// TIA Portal project "SistemRotativCuve_V19" (V19)

(* hardware
DEVICE "ET 200SP station_1"  ET 200SP-Station
   slot 0: "Rack_0"  Rack  6ES5 710-8MAx1
   slot 1: "PLC_1"  CPU 1510SP-1 PN  6ES7 510-1DK03-0AB0  V3.0
      slot 32768: "PROFINET interface_1"  X1
         slot 32771: "Port_3"  X1 P3
   slot 2: "DI 16x24VDC ST_1"  DI 16x24VDC ST  6ES7 131-6BH01-0BA0  V0.0
      slot 1: "DI 16x24VDC ST_1"  DI 16x24VDC ST
   slot 3: "DQ 16x24VDC/0.5A ST_1"  DQ 16x24VDC/0.5A ST  6ES7 132-6BH01-0BA0  V0.0
      slot 1: "DQ 16x24VDC/0.5A ST_1"  DQ 16x24VDC/0.5A ST
   slot 4: "Server module_1"  Server module  6ES7 193-6PA00-0AA0  V1.1
      slot 1: "Server module_1"  Server module
   slot 127: "BA 2xRJ45"  BA 2xRJ45  6ES7 193-6AR00-0AA0  V0.0
      slot 32769: "Port_1"  X1 P1  6ES7 193-6AR00-0AA0
      slot 32770: "Port_2"  X1 P2  6ES7 193-6AR00-0AA0
DEVICE "HMI_2"  KTP1200 Basic PN
   slot 0: "HMI_2"  KTP1200 Basic PN  6AV2 123-2MB03-0AX0  17.0.0.0
   slot 1: "HMI_RT_2"  KTP1200 Basic PN  6AV2 123-2MB03-0AX0  17.0.0.0
   slot 5: "HMI_2.IE_CP_1"  PROFINET Interface  17.0.0.0
      slot 1: "PROFINET Interface_1"  PROFINET Interface
         slot 1: "Port_1"  Port
*)

// ===== PLC "PLC_1"  CPU 1510SP-1 PN =====

VAR_GLOBAL   // PLC tag table "Default tag table"
   "System_Byte" AT %MB1 : Byte;
   "FirstScan" AT %M1.0 : Bool;
   "DiagStatusUpdate" AT %M1.1 : Bool;
   "AlwaysTRUE" AT %M1.2 : Bool;
   "AlwaysFALSE" AT %M1.3 : Bool;
END_VAR

VAR_GLOBAL   // PLC tag table "Clock Memory"
   "Clock_Byte" AT %MB0 : Byte;
   "Clock_10Hz" AT %M0.0 : Bool;
   "Clock_5Hz" AT %M0.1 : Bool;
   "Clock_2.5Hz" AT %M0.2 : Bool;
   "Clock_2Hz" AT %M0.3 : Bool;
   "Clock_1.25Hz" AT %M0.4 : Bool;
   "Clock_1Hz" AT %M0.5 : Bool;
   "Clock_0.625Hz" AT %M0.6 : Bool;
   "Clock_0.5Hz" AT %M0.7 : Bool;
END_VAR

VAR_GLOBAL   // PLC tag table "Motor_Tags"
   "Motor_Start" AT %M4.1 : Bool;
   "Motor_Stop" AT %M4.2 : Bool;
   "Motor_Ready_to_Start" AT %M4.3 : Bool;
END_VAR

VAR_GLOBAL   // PLC tag table "Sensors_Tags"
   "Barrier_Detection_Sensor1" AT %M3.0 : Bool;
   "Filling_Box_Sensor1" AT %M3.1 : Bool;
   "Emptying_Box_Sensor2" AT %M3.2 : Bool;
   "Barrier_Detection_Time_ON" AT %QD3 : DInt;
END_VAR

VAR_GLOBAL   // PLC tag table "Conveyor_Tags"
   "Conveyor_Start" AT %M5.1 : Bool;
   "Conveyor_Stop" AT %M5.2 : Bool;
   "Conveyor_Ready_to_Start" AT %M5.3 : Bool;
END_VAR

VAR_GLOBAL   // PLC tag table "Buttons"
   "Reset_Rotation_Counter" AT %M2.3 : Bool;
   "Switch_Manual_Mode_Position" AT %M2.4 : Bool;
   "One_Rotation_Move_Button" AT %M2.5 : Bool;
   "Switch_Automatic_Mode_Position" AT %M2.6 : Bool;
   "Switch_Stop_Mode_Position" AT %M2.7 : Bool;
END_VAR

VAR_GLOBAL   // PLC tag table "States"
   "Filled_All_Boxes" AT %M1.6 : Bool;
   "General_Stop_All_Filled" AT %M2.0 : Bool;
   "Automatic_Mode_ON" AT %M1.7 : Bool;
   "Manual_Mode_ON" AT %M2.1 : Bool;
   "General_Stop_Mode_ON" AT %M2.2 : Bool;
END_VAR

// folder: Conveyor/Data_Blocks

DATA_BLOCK "Conveyor_Drive_DB"   // DB4
{ S7_Optimized_Access := 'TRUE' }
VERSION : 0.1
// stored: InstanceOfName Conveyor_Drive_FB
"Conveyor_Drive_FB"
BEGIN
END_DATA_BLOCK

// folder: Motor/Data_Blocks

DATA_BLOCK "Counter_Box_Rotation_DB"   // DB2
{ S7_Optimized_Access := 'TRUE' }
AUTHOR : Simatic
FAMILY : IEC
NAME : CNTR
VERSION : 1.0
// stored: InstanceOfName IEC_COUNTER
"IEC_COUNTER"
BEGIN
END_DATA_BLOCK

DATA_BLOCK "Motor_Drive_DB"   // DB3
{ S7_Optimized_Access := 'TRUE' }
VERSION : 0.1
// stored: InstanceOfName Motor_Drive_FB
"Motor_Drive_FB"
BEGIN
END_DATA_BLOCK

// folder: Sensors/Data_Blocks

DATA_BLOCK "Validate_by_Sensors_DB"   // DB1
{ S7_Optimized_Access := 'TRUE' }
VERSION : 0.1
// stored: InstanceOfName Validate_by_Sensors_FB
"Validate_by_Sensors_FB"
BEGIN
END_DATA_BLOCK

DATA_BLOCK "IEC_Timer_0_DB"   // DB8
{ S7_Optimized_Access := 'TRUE' }
AUTHOR : Simatic
FAMILY : IEC
NAME : IEC_TMR
VERSION : 1.0
// stored: InstanceOfName IEC_TIMER
"IEC_TIMER"
BEGIN
END_DATA_BLOCK

// folder: Work Mode/Data_Blocks

DATA_BLOCK "Atomatic_Mode_DB"   // DB5
{ S7_Optimized_Access := 'TRUE' }
VERSION : 0.1
// stored: InstanceOfName Atomatic_Mode_FB
"Atomatic_Mode_FB"
BEGIN
END_DATA_BLOCK

DATA_BLOCK "Manual_Mode_DB"   // DB6
{ S7_Optimized_Access := 'TRUE' }
VERSION : 0.1
// stored: InstanceOfName Manual_Mode_FB
"Manual_Mode_FB"
BEGIN
END_DATA_BLOCK

DATA_BLOCK "General_Stop_Mode_DB"   // DB7
{ S7_Optimized_Access := 'TRUE' }
VERSION : 0.1
// stored: InstanceOfName General_Stop_Mode_FB
"General_Stop_Mode_FB"
BEGIN
END_DATA_BLOCK

// folder: (top level)

ORGANIZATION_BLOCK "Main"   // OB1, LAD, ProgramCycle
TITLE = "Main Program Sweep (Cycle)"
{ S7_Optimized_Access := 'TRUE' }
VERSION : 0.1
// Proiect realizat de Octavian Duma
   VAR_INPUT
      Initial_Call : Bool;   // Initial call of this OB
      Remanence : Bool;   // =True, if remanent data are available
   END_VAR
BEGIN

REGION Network 1: Automatic Mode enabled
   // Aici e scrisa logica de intrare in mod automat prin butonul cu 3 pozitii, setat pe pozitia de mod automat
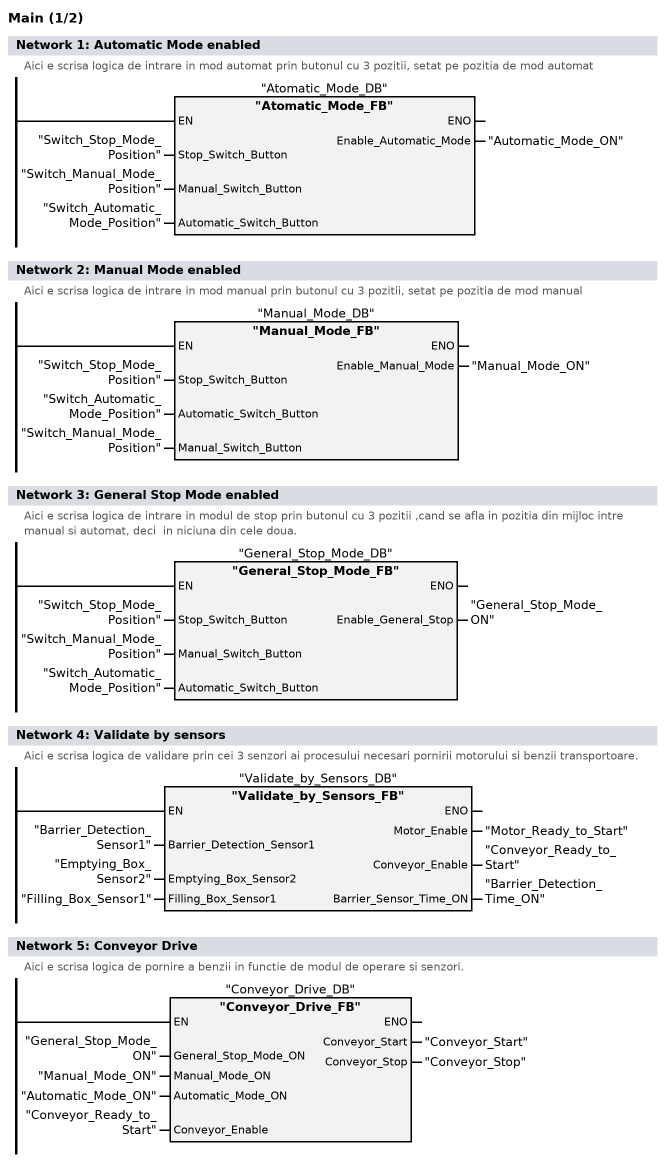
   RUNG wire#powerrail
      "Atomatic_Mode_DB"(Stop_Switch_Button := "Switch_Stop_Mode_Position", Manual_Switch_Button := "Switch_Manual_Mode_Position", Automatic_Switch_Button := "Switch_Automatic_Mode_Position", Enable_Automatic_Mode => "Automatic_Mode_ON")
   END_RUNG
   // the same network as SCL:
   "Atomatic_Mode_DB"(Stop_Switch_Button := "Switch_Stop_Mode_Position",   // "Atomatic_Mode_FB"
                      Manual_Switch_Button := "Switch_Manual_Mode_Position",
                      Automatic_Switch_Button := "Switch_Automatic_Mode_Position",
                      Enable_Automatic_Mode => "Automatic_Mode_ON");
END_REGION

REGION Network 2: Manual Mode enabled
   // Aici e scrisa logica de intrare in mod manual prin butonul cu 3 pozitii, setat pe pozitia de mod manual
   RUNG wire#powerrail
      "Manual_Mode_DB"(Stop_Switch_Button := "Switch_Stop_Mode_Position", Automatic_Switch_Button := "Switch_Automatic_Mode_Position", Manual_Switch_Button := "Switch_Manual_Mode_Position", Enable_Manual_Mode => "Manual_Mode_ON")
   END_RUNG
   // the same network as SCL:
   "Manual_Mode_DB"(Stop_Switch_Button := "Switch_Stop_Mode_Position",   // "Manual_Mode_FB"
                    Automatic_Switch_Button := "Switch_Automatic_Mode_Position",
                    Manual_Switch_Button := "Switch_Manual_Mode_Position",
                    Enable_Manual_Mode => "Manual_Mode_ON");
END_REGION

REGION Network 3: General Stop Mode enabled
   // Aici e scrisa logica de intrare in modul de stop prin butonul cu 3 pozitii ,cand se afla in pozitia din mijloc intre manual si automat, deci  in niciuna din cele doua.
   RUNG wire#powerrail
      "General_Stop_Mode_DB"(Stop_Switch_Button := "Switch_Stop_Mode_Position", Manual_Switch_Button := "Switch_Manual_Mode_Position", Automatic_Switch_Button := "Switch_Automatic_Mode_Position", Enable_General_Stop => "General_Stop_Mode_ON")
   END_RUNG
   // the same network as SCL:
   "General_Stop_Mode_DB"(Stop_Switch_Button := "Switch_Stop_Mode_Position",   // "General_Stop_Mode_FB"
                          Manual_Switch_Button := "Switch_Manual_Mode_Position",
                          Automatic_Switch_Button := "Switch_Automatic_Mode_Position",
                          Enable_General_Stop => "General_Stop_Mode_ON");
END_REGION

REGION Network 4: Validate by sensors
   // Aici e scrisa logica de validare prin cei 3 senzori ai procesului necesari pornirii motorului si benzii transportoare.
   RUNG wire#powerrail
      "Validate_by_Sensors_DB"(Barrier_Detection_Sensor1 := "Barrier_Detection_Sensor1", Emptying_Box_Sensor2 := "Emptying_Box_Sensor2", Filling_Box_Sensor1 := "Filling_Box_Sensor1", Motor_Enable => "Motor_Ready_to_Start", Conveyor_Enable => "Conveyor_Ready_to_Start", Barrier_Sensor_Time_ON => "Barrier_Detection_Time_ON")
   END_RUNG
   // the same network as SCL:
   "Validate_by_Sensors_DB"(Barrier_Detection_Sensor1 := "Barrier_Detection_Sensor1",   // "Validate_by_Sensors_FB"
                           Emptying_Box_Sensor2 := "Emptying_Box_Sensor2",
                           Filling_Box_Sensor1 := "Filling_Box_Sensor1",
                           Motor_Enable => "Motor_Ready_to_Start",
                           Conveyor_Enable => "Conveyor_Ready_to_Start",
                           Barrier_Sensor_Time_ON => "Barrier_Detection_Time_ON");
END_REGION

REGION Network 5: Conveyor Drive
   // Aici e scrisa logica de pornire a benzii in functie de modul de operare si senzori.
   RUNG wire#powerrail
      "Conveyor_Drive_DB"(General_Stop_Mode_ON := "General_Stop_Mode_ON", Manual_Mode_ON := "Manual_Mode_ON", Automatic_Mode_ON := "Automatic_Mode_ON", Conveyor_Enable := "Conveyor_Ready_to_Start", Conveyor_Start => "Conveyor_Start", Conveyor_Stop => "Conveyor_Stop")
   END_RUNG
   // the same network as SCL:
   "Conveyor_Drive_DB"(General_Stop_Mode_ON := "General_Stop_Mode_ON",   // "Conveyor_Drive_FB"
                       Manual_Mode_ON := "Manual_Mode_ON",
                       Automatic_Mode_ON := "Automatic_Mode_ON",
                       Conveyor_Enable := "Conveyor_Ready_to_Start",
                       Conveyor_Start => "Conveyor_Start",
                       Conveyor_Stop => "Conveyor_Stop");
END_REGION

REGION Network 6: Motor Drive
   // Aici e scrisa logica de pornire a motorului in functie de modul de operare, senzori, precum si cazul in care sistemul este plin complet si se goleste la buton in modul manual.
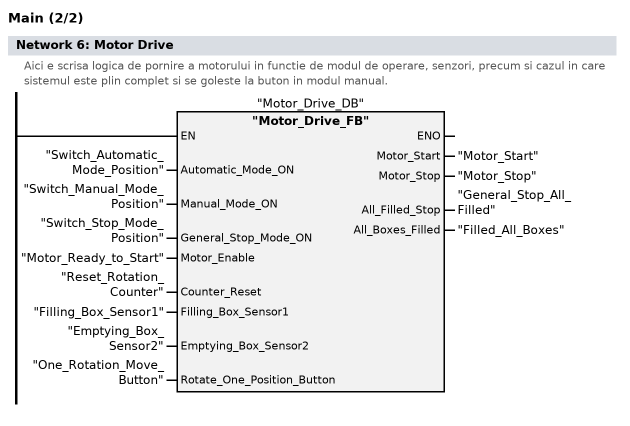
   RUNG wire#powerrail
      "Motor_Drive_DB"(Automatic_Mode_ON := "Switch_Automatic_Mode_Position", Manual_Mode_ON := "Switch_Manual_Mode_Position", General_Stop_Mode_ON := "Switch_Stop_Mode_Position", Motor_Enable := "Motor_Ready_to_Start", Counter_Reset := "Reset_Rotation_Counter", Filling_Box_Sensor1 := "Filling_Box_Sensor1", Emptying_Box_Sensor2 := "Emptying_Box_Sensor2", Rotate_One_Position_Button := "One_Rotation_Move_Button", Motor_Start => "Motor_Start", Motor_Stop => "Motor_Stop", All_Filled_Stop => "General_Stop_All_Filled", All_Boxes_Filled => "Filled_All_Boxes")
   END_RUNG
   // the same network as SCL:
   "Motor_Drive_DB"(Automatic_Mode_ON := "Switch_Automatic_Mode_Position",   // "Motor_Drive_FB"
                    Manual_Mode_ON := "Switch_Manual_Mode_Position",
                    General_Stop_Mode_ON := "Switch_Stop_Mode_Position",
                    Motor_Enable := "Motor_Ready_to_Start",
                    Counter_Reset := "Reset_Rotation_Counter",
                    Filling_Box_Sensor1 := "Filling_Box_Sensor1",
                    Emptying_Box_Sensor2 := "Emptying_Box_Sensor2",
                    Rotate_One_Position_Button := "One_Rotation_Move_Button",
                    Motor_Start => "Motor_Start",
                    Motor_Stop => "Motor_Stop",
                    All_Filled_Stop => "General_Stop_All_Filled",
                    All_Boxes_Filled => "Filled_All_Boxes");
END_REGION
END_ORGANIZATION_BLOCK

// folder: Conveyor/FunctionsDB

FUNCTION_BLOCK "Conveyor_Drive_FB"   // FB2, LAD
{ S7_Optimized_Access := 'TRUE' }
VERSION : 0.1
   VAR_INPUT
      General_Stop_Mode_ON : Bool;
      Manual_Mode_ON : Bool;
      Automatic_Mode_ON : Bool;
      Conveyor_Enable : Bool;
   END_VAR
   VAR_OUTPUT
      Conveyor_Start : Bool;
      Conveyor_Stop : Bool;
   END_VAR
BEGIN

REGION Network 1: Automatic Mode Conveyor is started
   // Banda este pornita in modul automat cand primeste semnalul de enable de la senzori.
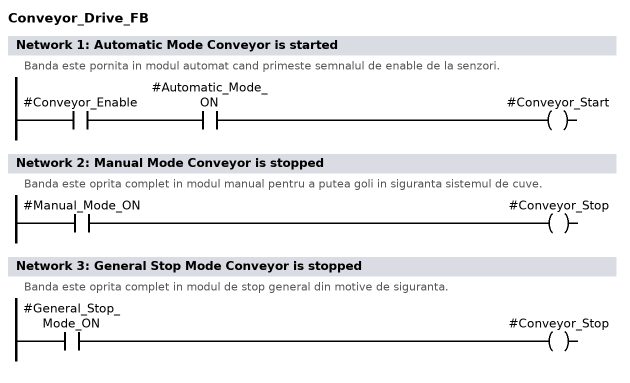
   RUNG wire#powerrail
      Contact( #Conveyor_Enable )
      Contact( #Automatic_Mode_ON )
      Coil( #Conveyor_Start )
   END_RUNG
   // the same network as SCL:
   #Conveyor_Start := #Conveyor_Enable AND #Automatic_Mode_ON;
END_REGION

REGION Network 2: Manual Mode Conveyor is stopped
   // Banda este oprita complet in modul manual pentru a putea goli in siguranta sistemul de cuve.
   RUNG wire#powerrail
      Contact( #Manual_Mode_ON )
      Coil( #Conveyor_Stop )
   END_RUNG
   // the same network as SCL:
   #Conveyor_Stop := #Manual_Mode_ON;
END_REGION

REGION Network 3: General Stop Mode Conveyor is stopped
   // Banda este oprita complet in modul de stop general din motive de siguranta.
   RUNG wire#powerrail
      Contact( #General_Stop_Mode_ON )
      Coil( #Conveyor_Stop )
   END_RUNG
   // the same network as SCL:
   #Conveyor_Stop := #General_Stop_Mode_ON;
END_REGION
END_FUNCTION_BLOCK

// folder: Motor/FunctionsDB

FUNCTION_BLOCK "Motor_Drive_FB"   // FB3, LAD
{ S7_Optimized_Access := 'TRUE' }
VERSION : 0.1
   VAR_INPUT
      Automatic_Mode_ON : Bool;
      Manual_Mode_ON : Bool;
      General_Stop_Mode_ON : Bool;
      Motor_Enable : Bool;
      Counter_Reset : Bool;
      Filling_Box_Sensor1 : Bool;
      Emptying_Box_Sensor2 : Bool;
      Rotate_One_Position_Button : Bool;
   END_VAR
   VAR_OUTPUT
      Motor_Start : Bool;
      Motor_Stop : Bool;
      All_Filled_Stop : Bool;
      All_Boxes_Filled : Bool;
   END_VAR
   VAR
      Rotation_Command : Bool;
   END_VAR
BEGIN

REGION Network 1: Manual Mode Rotation Command
   // Comanda de rotire manuala cu cate o pozitie a cuvei este conditionata de modul manual si de apasarea butonului fizic de pe panoul de comanda.
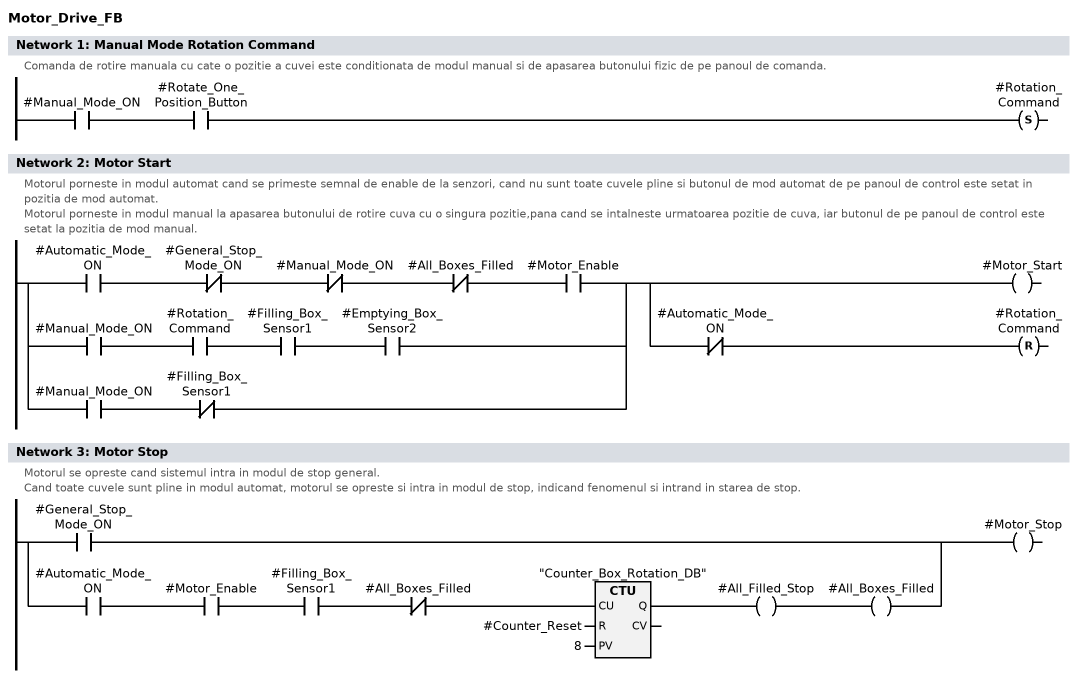
   RUNG wire#powerrail
      Contact( #Manual_Mode_ON )
      Contact( #Rotate_One_Position_Button )
      S_Coil( #Rotation_Command )
   END_RUNG
   // the same network as SCL:
   IF #Manual_Mode_ON AND #Rotate_One_Position_Button THEN #Rotation_Command := TRUE; END_IF;
END_REGION

REGION Network 2: Motor Start
   // Motorul porneste in modul automat cand se primeste semnal de enable de la senzori, cand nu sunt toate cuvele pline si butonul de mod automat de pe panoul de control este setat in pozitia de mod automat. 
   //       Motorul porneste in modul manual la apasarea butonului de rotire cuva cu o singura pozitie,pana cand se intalneste urmatoarea pozitie de cuva, iar butonul de pe panoul de control este setat la pozitia de mod manual.
   RUNG wire#powerrail
      Contact( #Automatic_Mode_ON )
      I_Contact( #General_Stop_Mode_ON )
      I_Contact( #Manual_Mode_ON )
      I_Contact( #All_Boxes_Filled )
      Contact( #Motor_Enable )
      wire#w1
      Coil( #Motor_Start )
   END_RUNG
   RUNG wire#powerrail
      Contact( #Manual_Mode_ON )
      Contact( #Rotation_Command )
      Contact( #Filling_Box_Sensor1 )
      Contact( #Emptying_Box_Sensor2 )
   END_RUNG wire#w1
   RUNG wire#powerrail
      Contact( #Manual_Mode_ON )
      I_Contact( #Filling_Box_Sensor1 )
   END_RUNG wire#w1
   RUNG wire#w1
      I_Contact( #Automatic_Mode_ON )
      R_Coil( #Rotation_Command )
   END_RUNG
   // the same network as SCL:
   #Motor_Start := (#Automatic_Mode_ON AND NOT #General_Stop_Mode_ON AND NOT #Manual_Mode_ON AND NOT #All_Boxes_Filled AND #Motor_Enable) OR (#Manual_Mode_ON AND #Rotation_Command AND #Filling_Box_Sensor1 AND #Emptying_Box_Sensor2) OR (#Manual_Mode_ON AND NOT #Filling_Box_Sensor1);
   IF #Motor_Start AND NOT #Automatic_Mode_ON THEN #Rotation_Command := FALSE; END_IF;
END_REGION

REGION Network 3: Motor Stop
   // Motorul se opreste cand sistemul intra in modul de stop general.
   // Cand toate cuvele sunt pline in modul automat, motorul se opreste si intra in modul de stop, indicand fenomenul si intrand in starea de stop.
   "Counter_Box_Rotation_DB".CTU(CU := #Automatic_Mode_ON AND #Motor_Enable AND #Filling_Box_Sensor1 AND NOT #All_Boxes_Filled,
                           R := #Counter_Reset,
                           PV := 8);
   #All_Filled_Stop := "Counter_Box_Rotation_DB".Q;
   #All_Boxes_Filled := "Counter_Box_Rotation_DB".Q;
   #Motor_Stop := #General_Stop_Mode_ON OR "Counter_Box_Rotation_DB".Q;
END_REGION
END_FUNCTION_BLOCK

// folder: Sensors/FunctionsDB

FUNCTION_BLOCK "Validate_by_Sensors_FB"   // FB1, LAD
{ S7_Optimized_Access := 'TRUE' }
VERSION : 0.1
   VAR_INPUT
      Barrier_Detection_Sensor1 : Bool;
      Emptying_Box_Sensor2 : Bool;
      Filling_Box_Sensor1 : Bool;
   END_VAR
   VAR_OUTPUT
      Motor_Enable : Bool;
      Conveyor_Enable : Bool;
      Barrier_Sensor_Time_ON : DInt;
   END_VAR
   VAR
      Filled_Box : Bool;
   END_VAR
BEGIN

REGION Network 1: A box is full when barrier sensor is ON for 5 seconds
   // Logica de verificare a semnalului senzorului. Pentru a evita activarea conditiei de cuva plina de catre suruburile care cad in cuva de pe banda, senzorul va trebui sa fie activ cel putin 5 secunde ca sa consideram atingerea nivelului de umplere.
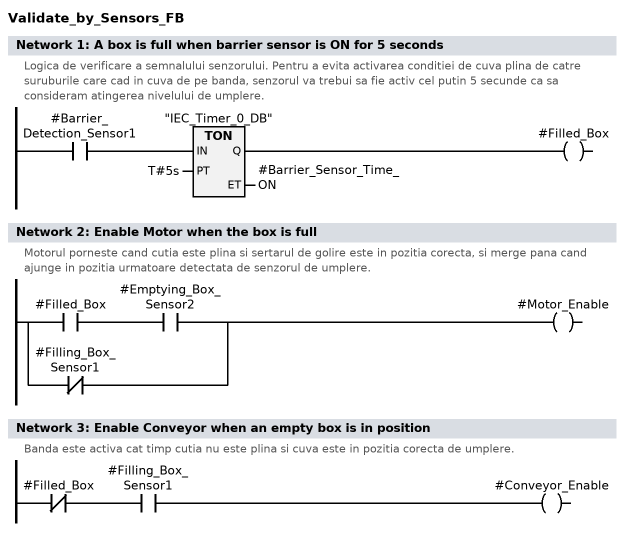
   "IEC_Timer_0_DB".TON(IN := #Barrier_Detection_Sensor1, PT := T#5s, ET => #Barrier_Sensor_Time_ON);
   #Filled_Box := "IEC_Timer_0_DB".Q;
END_REGION

REGION Network 2: Enable Motor when the box is full
   // Motorul porneste cand cutia este plina si sertarul de golire este in pozitia corecta, si merge pana cand ajunge in pozitia urmatoare detectata de senzorul de umplere.
   RUNG wire#powerrail
      Contact( #Filled_Box )
      Contact( #Emptying_Box_Sensor2 )
      wire#w1
      Coil( #Motor_Enable )
   END_RUNG
   RUNG wire#powerrail
      I_Contact( #Filling_Box_Sensor1 )
   END_RUNG wire#w1
   // the same network as SCL:
   #Motor_Enable := (#Filled_Box AND #Emptying_Box_Sensor2) OR NOT #Filling_Box_Sensor1;
END_REGION

REGION Network 3: Enable Conveyor when an empty box is in position
   // Banda este activa cat timp cutia nu este plina si cuva este in pozitia corecta de umplere.
   RUNG wire#powerrail
      I_Contact( #Filled_Box )
      Contact( #Filling_Box_Sensor1 )
      Coil( #Conveyor_Enable )
   END_RUNG
   // the same network as SCL:
   #Conveyor_Enable := NOT #Filled_Box AND #Filling_Box_Sensor1;
END_REGION
END_FUNCTION_BLOCK

// folder: Work Mode/FunctionsDB

FUNCTION_BLOCK "Atomatic_Mode_FB"   // FB4, LAD
{ S7_Optimized_Access := 'TRUE' }
VERSION : 0.1
   VAR_INPUT
      Stop_Switch_Button : Bool;
      Manual_Switch_Button : Bool;
      Automatic_Switch_Button : Bool;
   END_VAR
   VAR_OUTPUT
      Enable_Automatic_Mode : Bool;
   END_VAR
BEGIN

REGION Network 1: Enable Automatic Mode while other mode is disabled
   // Sistemul intra in modul automat pe baza switch-ului cu 3 pozitii, care va fi doar pe pozitia de mod automat , implicand ca celelalte pozitii sa fie dezactivate. Se tine cont si de faptul ca sistemul nu este oprit de umplerea tuturor cuvelor.
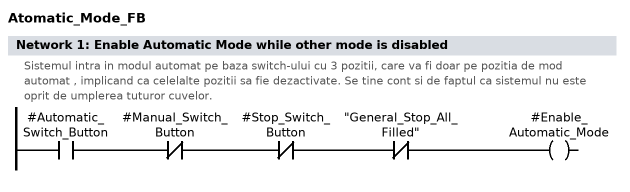
   RUNG wire#powerrail
      Contact( #Automatic_Switch_Button )
      I_Contact( #Manual_Switch_Button )
      I_Contact( #Stop_Switch_Button )
      I_Contact( "General_Stop_All_Filled" )
      Coil( #Enable_Automatic_Mode )
   END_RUNG
   // the same network as SCL:
   #Enable_Automatic_Mode := #Automatic_Switch_Button AND NOT #Manual_Switch_Button AND NOT #Stop_Switch_Button AND NOT "General_Stop_All_Filled";
END_REGION
END_FUNCTION_BLOCK

FUNCTION_BLOCK "Manual_Mode_FB"   // FB5, LAD
{ S7_Optimized_Access := 'TRUE' }
VERSION : 0.1
   VAR_INPUT
      Stop_Switch_Button : Bool;
      Automatic_Switch_Button : Bool;
      Manual_Switch_Button : Bool;
   END_VAR
   VAR_OUTPUT
      Enable_Manual_Mode : Bool;
   END_VAR
BEGIN

REGION Network 1: Enable Manual Mode while other mode is disabled
   // Sistemul intra in modul manual pe baza switch-ului cu 3 pozitii, care va fi doar pe pozitia de mod manual , implicand ca celelalte pozitii sa fie dezactivate. Se tine cont si de faptul ca sistemul nu este oprit de umplerea tuturor cuvelor.
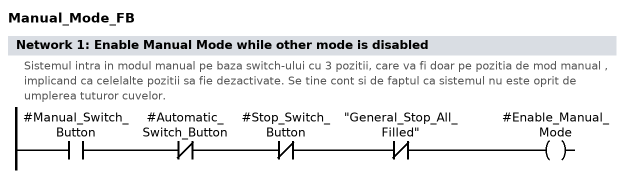
   RUNG wire#powerrail
      Contact( #Manual_Switch_Button )
      I_Contact( #Automatic_Switch_Button )
      I_Contact( #Stop_Switch_Button )
      I_Contact( "General_Stop_All_Filled" )
      Coil( #Enable_Manual_Mode )
   END_RUNG
   // the same network as SCL:
   #Enable_Manual_Mode := #Manual_Switch_Button AND NOT #Automatic_Switch_Button AND NOT #Stop_Switch_Button AND NOT "General_Stop_All_Filled";
END_REGION
END_FUNCTION_BLOCK

FUNCTION_BLOCK "General_Stop_Mode_FB"   // FB6, LAD
{ S7_Optimized_Access := 'TRUE' }
VERSION : 0.1
   VAR_INPUT
      Stop_Switch_Button : Bool;
      Manual_Switch_Button : Bool;
      Automatic_Switch_Button : Bool;
   END_VAR
   VAR_OUTPUT
      Enable_General_Stop : Bool;
   END_VAR
BEGIN

REGION Network 1: Enable General Stop Mode while other mode is disabled
   // Sistemul intra in modul automat pe baza switch-ului cu 3 pozitii, care va fi doar pe pozitia de mod general de stop, fiind pozitia de la mijloc,intre celelate moduri , implicand ca celelalte pozitii sa fie dezactivate.
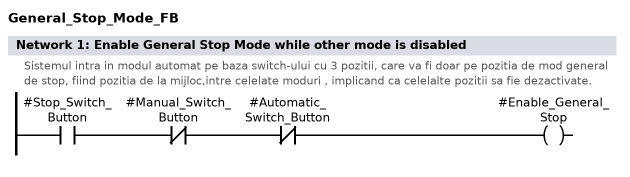
   RUNG wire#powerrail
      Contact( #Stop_Switch_Button )
      I_Contact( #Manual_Switch_Button )
      I_Contact( #Automatic_Switch_Button )
      Coil( #Enable_General_Stop )
   END_RUNG
   // the same network as SCL:
   #Enable_General_Stop := #Stop_Switch_Button AND NOT #Manual_Switch_Button AND NOT #Automatic_Switch_Button;
END_REGION
END_FUNCTION_BLOCK

(* ===== HMI "HMI_RT_2" =====
system functions are stored by id; their names below are inferred from use
connection "HMI_Connection_2": ETHERNET, SMART_S7_1500_OMS

HMI tags "Default tag table"
   "Tag_ScreenNumber" : UInt, internal
   "BarrierDetectionSensor1" : Bool = PLC Barrier_Detection_Sensor1 AT %M3.0, 1 s
   "Conveyor_Ready_to_Start" : Bool = PLC Conveyor_Ready_to_Start AT %M5.3, 1 s
   "Conveyor_Start" : Bool = PLC Conveyor_Start AT %M5.1, 1 s
   "Conveyor_Stop" : Bool = PLC Conveyor_Stop AT %M5.2, 1 s
   "EmptyingBoxSensor2" : Bool = PLC Emptying_Box_Sensor2 AT %M3.2, 1 s
   "FillingBoxSensor1" : Bool = PLC Filling_Box_Sensor1 AT %M3.1, 1 s
   "General_Stop_All_Filled" : Bool = PLC General_Stop_All_Filled AT %M2.0, 1 s
   "Motor_Ready_to_Start" : Bool = PLC Motor_Ready_to_Start AT %M4.3, 1 s
   "Motor_Start" : Bool = PLC Motor_Start AT %M4.1, 1 s
   "Motor_Stop" : Bool = PLC Motor_Stop AT %M4.2, 1 s
   "Reset_Rotation_Counter" : Bool = PLC Reset_Rotation_Counter AT %M2.3, 1 s
   "Rotation_Counter" : Int = PLC Counter_Box_Rotation_DB.CV AT %DB1.DBX0.0, 1 s
   "System_Full" : Bool = PLC Filled_All_Boxes AT %M1.6, 1 s
   "Automatic_Mode_Switch_Position" : Bool = PLC Switch_Automatic_Mode_Position AT %M2.6, 1 s
   "Automatic_Mode_ON" : Bool = PLC Automatic_Mode_ON AT %M1.7, 1 s
   "Manual_Mode_Swich_Position" : Bool = PLC Switch_Manual_Mode_Position AT %M2.4, 1 s
   "Manual_Mode_ON" : Bool = PLC Manual_Mode_ON AT %M2.1, 1 s
   "General_Stop_Swich_Position" : Bool = PLC Switch_Stop_Mode_Position AT %M2.7, 1 s
   "General_Stop_ON" : Bool = PLC General_Stop_Mode_ON AT %M2.2, 1 s
   "One_Step_Move_Button" : Bool = PLC One_Rotation_Move_Button AT %M2.5, 1 s
   "Barrier_Sensor_Timer_Value" : DInt = PLC Barrier_Detection_Time_ON AT %QD3, 1 s

Template "Template_1" 1280x800
   Button "Exit" at 1182,752 size 67x47; TextOff 'Exit'; PictureOff "ExitRuntime_KTP1200_Basic_PN_TR"; PictureOn "ExitRuntime_KTP1200_Basic_PN_TR"
      on Release: StopRuntime(0)
   Button "Language" at 1054,752 size 67x47; TextOff 'Language'; PictureOff "ToggleLanguage_KTP1200_Basic_PN_TR"; PictureOn "ToggleLanguage_KTP1200_Basic_PN_TR"
      on Release: function_fb9197e8(-1)
   Button "Template_Button" at 926,752 size 67x47; TextOff 'Text'
   Button "Template_Button_1" at 798,752 size 67x47; TextOff 'Text'
   Button "Template_Button_2" at 670,752 size 67x47; TextOff 'Text'
   Button "Template_Button_3" at 542,752 size 67x47; TextOff 'Text'
   Button "Template_Button_4" at 414,752 size 67x47; TextOff 'Text'
   Button "Template_Button_5" at 286,752 size 67x47; TextOff 'Text'
   Button "Alarms" at 158,752 size 67x47; TextOff 'Alarms'; PictureOff "AlarmDisplay_KTP1200_Basic_PN_TR"; PictureOn "AlarmDisplay_KTP1200_Basic_PN_TR"
      on Release: function_ef3f5d25("Alarm window_Unacknowledged", -1)
   Button "Start screen" at 30,752 size 67x47; TextOff 'Start screen'; PictureOff "NavigateHome_KTP1200_Basic_PN_TR"; PictureOn "NavigateHome_KTP1200_Basic_PN_TR"
      on Release: ActivateScreen("HMI Proces", 0)
   SymbolicIOField "Symbolic_IO_Field_Screen" at 87,9 size 1086x30; TextOff '0'; TextOn '1'; TextList "TextList_ScreenNames"
      ProcessValue <- "Tag_ScreenNumber"
      on Change: ActivateScreenByNumber("Tag_ScreenNumber", 0)
   DateTimeField "HmiScreenItemData" at 1175,24 size 105x24
   DateTimeField "HmiScreenItemData_1" at 1175,0 size 105x24
   GraphicView "Logo" at 0,0 size 85x48; Picture "Logo of HMI_2"

screen "HMI Proces" 1280x800, template "Template_1"
   on GenerateScreen: SetTag("Tag_ScreenNumber", 1)
   GraphicView "Graphic view_1" at 40,139 size 57x61; Picture "OJ5126"
   GraphicView "Graphic view_4" at 46,253 size 45x64; Picture "IE5338"
   TextField "Text field_1" at 16,106 size 119x21; Text 'Barrier Sensor'
   TextField "Text field_3" at 16,221 size 162x21; Text 'Filling Box Sensor 1'
   GraphicView "Graphic view_2" at 524,143 size 136x100; Picture "Motor_1"
   Rectangle "Rectangle_4" at 795,185 size 53x48
      Appearance <- "Motor_Start"
   TextField "Text field_5" at 524,106 size 59x25; Text 'Motor'
   GraphicView "Graphic view_3" at 524,316 size 136x100; Picture "banda"
   Rectangle "Rectangle_2" at 278,260 size 54x46
      Appearance <- "FillingBoxSensor1"
   Rectangle "Rectangle_1" at 277,152 size 54x46
      Appearance <- "BarrierDetectionSensor1"
   Rectangle "Rectangle_3" at 795,355 size 53x48
      Appearance <- "Conveyor_Start"
   TextField "Text field_2" at 16,325 size 189x21; Text 'Emptying Box Sensor 2'
   Rectangle "Rectangle_5" at 278,373 size 54x46
      Appearance <- "EmptyingBoxSensor2"
   TextField "Text field_6" at 524,281 size 92x25; Text 'Conveyor'
   Button "Button_1" at 136,139 size 93x61; TextOff 'Activate'
      on Press: InvertBit("BarrierDetectionSensor1")
      Appearance <- "BarrierDetectionSensor1"
   Button "Button_2" at 136,253 size 92x60; TextOff 'Activate'
      on Press: InvertBit("FillingBoxSensor1")
      Appearance <- "FillingBoxSensor1"
   Button "Button_3" at 136,367 size 91x59; TextOff 'Activate'
      on Press: InvertBit("EmptyingBoxSensor2")
      Appearance <- "EmptyingBoxSensor2"
   Button "Button_4" at 907,552 size 175x55; TextOff 'RESET'
      on Press: function_b14e0dd5("Reset_Rotation_Counter", 0)
      Appearance <- "Reset_Rotation_Counter"
   Circle "Circle_1" at 297,552 size 60x60
      Appearance <- "General_Stop_All_Filled"
   TextField "Text field_7" at 120,651 size 127x21; Text 'All Boxes is full'
   TextField "Text field_8" at 278,651 size 108x21; Text 'General Stop'
   Circle "Circle_2" at 153,554 size 61x61
      Appearance <- "System_Full"
   Circle "Circle_3" at 440,552 size 60x60
      Appearance <- "General_Stop_All_Filled"
   TextField "Text field_9" at 419,650 size 105x21; Text 'Process RUN'
   Circle "Circle_4" at 701,177 size 65x65
      Appearance <- "Motor_Ready_to_Start"
   Circle "Circle_5" at 697,348 size 66x66
      Appearance <- "Conveyor_Ready_to_Start"
   TextField "Text field_10" at 705,312 size 53x21; Text 'Ready'
   TextField "Text field_11" at 705,142 size 53x21; Text 'Ready'
   IOField "I/O field_1" at 570,555 size 61x53; FormatPattern 9
      ProcessValue <- "Rotation_Counter"
   GraphicView "Graphic view_6" at 46,362 size 45x64; Picture "IE5338"
   TextField "Text field_4" at 277,127 size 50x25; Text 'State'
   TextField "Text field_12" at 793,142 size 50x25; Text 'State'
   TextField "Text field_13" at 793,316 size 50x25; Text 'State'
   TextField "Text field_14" at 277,230 size 50x25; Text 'State'
   TextField "Text field_15" at 277,342 size 50x25; Text 'State'
   TextField "Text field_16" at 544,648 size 110x23; Text 'Box Number'
   TextField "Text field_17" at 962,55 size 228x43; Text 'System Mode'
   Button "Button_5" at 953,214 size 130x46; TextOff 'AUTOMATIC'
      on Press: InvertBit("Automatic_Mode_Switch_Position")
      Appearance <- "Automatic_Mode_Switch_Position"
   Button "Button_6" at 952,293 size 130x46; TextOff 'MANUAL'
      on Press: InvertBit("Manual_Mode_Swich_Position")
      Appearance <- "Manual_Mode_Swich_Position"
   Button "Button_7" at 952,139 size 130x46; TextOff 'STOP'
      on Press: InvertBit("General_Stop_Swich_Position")
      Appearance <- "General_Stop_Swich_Position"
   Rectangle "Rectangle_6" at 1123,224 size 35x31
      Appearance <- "Automatic_Mode_ON"
   Rectangle "Rectangle_7" at 1123,298 size 36x31
      Appearance <- "Manual_Mode_ON"
   Rectangle "Rectangle_8" at 1124,149 size 35x31
      Appearance <- "General_Stop_ON"
   Button "Button_8" at 952,369 size 114x34; TextOff 'ROTATE'
      on Press: function_b14e0dd5("One_Step_Move_Button", 0)
      Appearance <- "One_Step_Move_Button"
   TextField "Text field_19" at 278,470 size 231x43; Text 'System States'
   TextField "Text field_20" at 136,52 size 148x43; Text 'Sensors'
   TextField "Text field_21" at 625,52 size 159x43; Text 'Actuators'
   TextField "Text field_23" at 878,470 size 221x43; Text 'System Reset'
   TextField "Text field_24" at 1169,230 size 50x25; Text 'State'
   TextField "Text field_25" at 1168,304 size 50x25; Text 'State'
   TextField "Text field_26" at 1169,160 size 50x25; Text 'State'
   TextField "Text field_27" at 1083,378 size 136x25; Text 'Rotate one box'
   IOField "I/O field_2" at 373,163 size 59x32; FormatPattern 9999
      ProcessValue <- "Barrier_Sensor_Timer_Value"
   TextField "Text field_22" at 381,141 size 41x22; Text 'Time'
   TextField "Text field_28" at 364,127 size 81x22; Text 'Activation'
   TextField "Text field_18" at 204,14 size 386x22; Text 'AUTOMATED SCREW TANK FILLING SYSTEM MENU'
*)